// TIA Portal project "SortingStation" (V19)

(* hardware
DEVICE "S71500/ET200MP-Station_1"  S7-1500 station
   slot 0: "Profilschiene_0"  6ES7 590-1***0-0AA0
   slot 1: "PLC_1"  CPU 1511-1 PN  6ES7 511-1AK00-0AB0  V1.8
   slot 2: "AI 8xU/I/RTD/TC ST_1"  AI 8xU/I/RTD/TC ST  6ES7 531-7KF00-0AB0  V2.0
   slot 3: "AI 8xU/I/RTD/TC ST_2"  AI 8xU/I/RTD/TC ST  6ES7 531-7KF00-0AB0  V2.0
   slot 4: "AI 8xU/I/RTD/TC ST_3"  AI 8xU/I/RTD/TC ST  6ES7 531-7KF00-0AB0  V2.0
   slot 5: "AI 8xU/I/RTD/TC ST_4"  AI 8xU/I/RTD/TC ST  6ES7 531-7KF00-0AB0  V2.0
   slot 6: "DI 16x24VDC BA_1"  DI 16x24VDC BA  6ES7 521-1BH10-0AA0  V1.0
*)

// ===== PLC "PLC_1"  CPU 1511-1 PN =====

VAR_GLOBAL   // PLC tag table "Standard-Variablentabelle"
   "Tag_1" AT %I1.1 : Bool;
   "Tag_2" AT %Q1.6 : Bool;
   "Tag_3" AT %I1.2 : Bool;
END_VAR

VAR_GLOBAL   // PLC tag table "Tag table_1"
   "At exit" AT %I0.0 : Bool;
   "Start" AT %I0.1 : Bool;
   "Reset" AT %I0.2 : Bool;
   "Stop" AT %I0.3 : Bool;
   "Emergency stop" AT %I0.4 : Bool;
   "Auto" AT %I0.5 : Bool;
   "FACTORY I/O (Running)" AT %I0.6 : Bool;
   "Entry conveyor" AT %Q0.0 : Bool;
   "Stop blade" AT %Q0.1 : Bool;
   "Exit conveyor" AT %Q0.2 : Bool;
   "Sorter 1 turn" AT %Q0.3 : Bool;
   "Sorter 1 belt" AT %Q0.4 : Bool;
   "Sorter 2 turn" AT %Q0.5 : Bool;
   "Sorter 2 belt" AT %Q0.6 : Bool;
   "Sorter 3 turn" AT %Q0.7 : Bool;
   "Sorter 3 belt" AT %Q1.0 : Bool;
   "Start light" AT %Q1.1 : Bool;
   "Reset light" AT %Q1.2 : Bool;
   "Stop light" AT %Q1.3 : Bool;
   "Counter 1" AT %QD30 : DInt;
   "Counter 2" AT %QD34 : DInt;
   "Counter 3" AT %QD38 : DInt;
   "Vision sensor" AT %ID30 : DInt;
   "BoxLeft" AT %M0.1 : Bool;
   "BoxLeft2" AT %M0.2 : Bool;
   "BoxLeft3" AT %M0.4 : Bool;
   "SensorEdgeMem" AT %M0.0 : Bool;
   "BoxLeftStopBlade" AT %M0.3 : Bool;
   "Emitter" AT %Q1.4 : Bool;
END_VAR

DATA_BLOCK "EntryConveyor_DB"   // DB2
{ S7_Optimized_Access := 'TRUE' }
VERSION : 0.1
// stored: InstanceOfName Entry/ExitConveyor
"Entry/ExitConveyor"
BEGIN
END_DATA_BLOCK

DATA_BLOCK "Start/Stop_DB"   // DB3
{ S7_Optimized_Access := 'TRUE' }
VERSION : 0.1
// stored: InstanceOfName Start/Stop
"Start/Stop"
BEGIN
END_DATA_BLOCK

DATA_BLOCK "Stopblade_DB"   // DB4
{ S7_Optimized_Access := 'TRUE' }
VERSION : 0.1
// stored: InstanceOfName Stopblade
"Stopblade"
BEGIN
END_DATA_BLOCK

DATA_BLOCK "Sorter1_DB_1"   // DB5
{ S7_Optimized_Access := 'TRUE' }
VERSION : 0.1
// stored: InstanceOfName Sorter1
"Sorter1"
BEGIN
END_DATA_BLOCK

DATA_BLOCK "Sorter2_DB_1"   // DB8
{ S7_Optimized_Access := 'TRUE' }
VERSION : 0.1
// stored: InstanceOfName Sorter2
"Sorter2"
BEGIN
END_DATA_BLOCK

DATA_BLOCK "Sorter3_DB_1"   // DB9
{ S7_Optimized_Access := 'TRUE' }
VERSION : 0.1
// stored: InstanceOfName Sorter3
"Sorter3"
BEGIN
END_DATA_BLOCK

DATA_BLOCK "Counters_DB"   // DB11
{ S7_Optimized_Access := 'TRUE' }
VERSION : 0.1
// stored: InstanceOfName Counters
"Counters"
BEGIN
END_DATA_BLOCK

// folder: System blocks/Program resources

DATA_BLOCK "IEC_Timer_0_DB"   // DB1
{ S7_Optimized_Access := 'TRUE' }
AUTHOR : Simatic
FAMILY : IEC
NAME : IEC_TMR
VERSION : 1.0
// stored: InstanceOfName IEC_TIMER
"IEC_TIMER"
BEGIN
   PT := T#250MS;
END_DATA_BLOCK

DATA_BLOCK "IEC_Counter_1_DB"   // DB6
{ S7_Optimized_Access := 'TRUE' }
AUTHOR : Simatic
FAMILY : IEC
NAME : CNTR
VERSION : 1.0
// stored: InstanceOfName IEC_COUNTER
"IEC_COUNTER"
BEGIN
   PV := 100;
END_DATA_BLOCK

DATA_BLOCK "IEC_Counter_0_DB_1"   // DB7
{ S7_Optimized_Access := 'TRUE' }
AUTHOR : Simatic
FAMILY : IEC
NAME : CNTR
VERSION : 1.0
// stored: InstanceOfName IEC_COUNTER
"IEC_COUNTER"
BEGIN
   PV := 100;
END_DATA_BLOCK

DATA_BLOCK "IEC_Counter_2_DB"   // DB10
{ S7_Optimized_Access := 'TRUE' }
AUTHOR : Simatic
FAMILY : IEC
NAME : CNTR
VERSION : 1.0
// stored: InstanceOfName IEC_COUNTER
"IEC_COUNTER"
BEGIN
   PV := 100;
END_DATA_BLOCK

// folder: (top level)

FUNCTION_BLOCK "Start/Stop"   // FB1, LAD
{ S7_Optimized_Access := 'TRUE' }
VERSION : 0.1
BEGIN

REGION Network 1
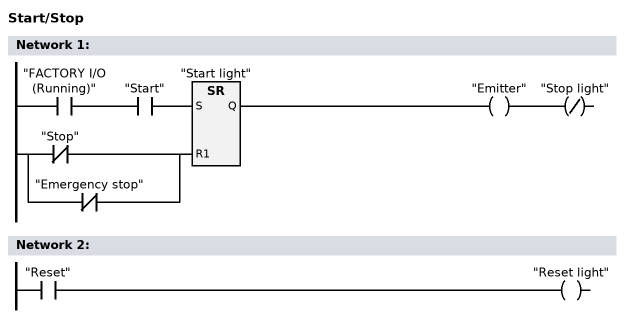
   RUNG wire#powerrail
      Contact( "FACTORY I/O (Running)" )
      Contact( "Start" )
      S_SR(operand := "Start light", r1 := wire#w1)
      Coil( "Emitter" )
      I_Coil( "Stop light" )
   END_RUNG
   RUNG wire#powerrail
      I_Contact( "Stop" )
   END_RUNG wire#w1
   RUNG wire#powerrail
      I_Contact( "Emergency stop" )
   END_RUNG wire#w1
   // the same network as SCL:
   IF "FACTORY I/O (Running)" AND "Start" THEN
       "Start light" := TRUE;   // SR flip-flop
   END_IF;
   IF NOT "Stop" OR NOT "Emergency stop" THEN "Start light" := FALSE; END_IF;
   "Emitter" := "Start light";
   "Stop light" := NOT "Start light";
END_REGION

REGION Network 2
   RUNG wire#powerrail
      Contact( "Reset" )
      Coil( "Reset light" )
   END_RUNG
   // the same network as SCL:
   "Reset light" := "Reset";
END_REGION
END_FUNCTION_BLOCK

FUNCTION_BLOCK "Sorter1"   // FB2, LAD
{ S7_Optimized_Access := 'TRUE' }
VERSION : 0.1
   VAR_TEMP   // added for the SCL form of the ladder/FBD networks
      _w1 : Bool;
   END_VAR
BEGIN

REGION Network 1
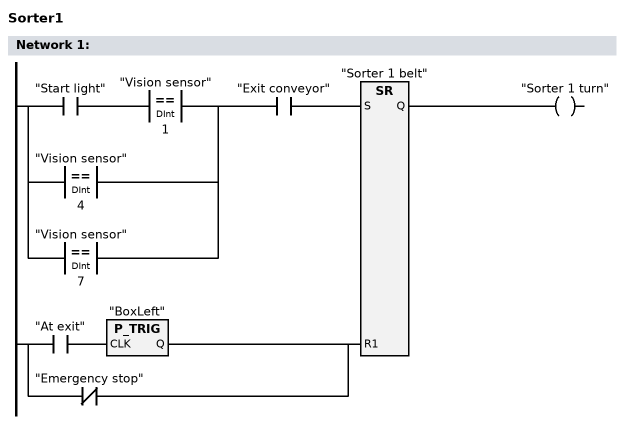
   RUNG wire#powerrail
      Contact( "Start light" )
      { S7_Templates := "SrcType := DInt" } EQ_Contact(in1 := "Vision sensor", in2 := 1)
      wire#w1
      Contact( "Exit conveyor" )
      S_SR(operand := "Sorter 1 belt", r1 := wire#w2)
      Coil( "Sorter 1 turn" )
   END_RUNG
   RUNG wire#powerrail
      { S7_Templates := "SrcType := DInt" } EQ_Contact(in1 := "Vision sensor", in2 := 4)
   END_RUNG wire#w1
   RUNG wire#powerrail
      { S7_Templates := "SrcType := DInt" } EQ_Contact(in1 := "Vision sensor", in2 := 7)
   END_RUNG wire#w1
   RUNG wire#powerrail
      Contact( "At exit" )
      P_Trig( "BoxLeft" )
   END_RUNG wire#w2
   RUNG wire#powerrail
      I_Contact( "Emergency stop" )
   END_RUNG wire#w2
   // the same network as SCL:
   #_w1 := "At exit" AND NOT "BoxLeft";   // rising edge
   "BoxLeft" := "At exit";
   IF (("Start light" AND ("Vision sensor" = 1)) OR ("Vision sensor" = 4) OR ("Vision sensor" = 7)) AND "Exit conveyor" THEN
       "Sorter 1 belt" := TRUE;   // SR flip-flop
   END_IF;
   IF #_w1 OR NOT "Emergency stop" THEN "Sorter 1 belt" := FALSE; END_IF;
   "Sorter 1 turn" := "Sorter 1 belt";
END_REGION
END_FUNCTION_BLOCK

FUNCTION_BLOCK "Sorter2"   // FB3, LAD
{ S7_Optimized_Access := 'TRUE' }
VERSION : 0.1
   VAR_TEMP   // added for the SCL form of the ladder/FBD networks
      _w1 : Bool;
   END_VAR
BEGIN

REGION Network 1
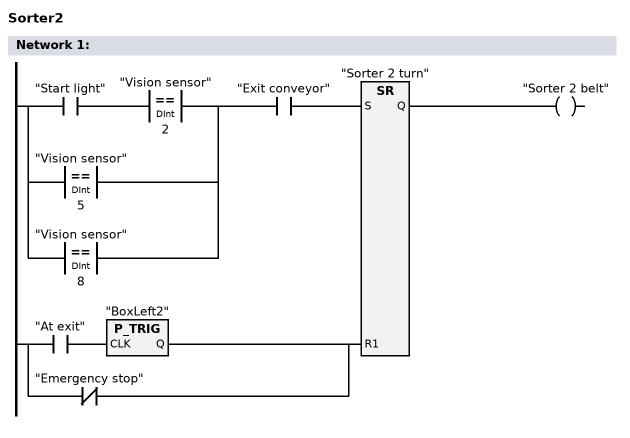
   RUNG wire#powerrail
      Contact( "Start light" )
      { S7_Templates := "SrcType := DInt" } EQ_Contact(in1 := "Vision sensor", in2 := 2)
      wire#w1
      Contact( "Exit conveyor" )
      S_SR(operand := "Sorter 2 turn", r1 := wire#w2)
      Coil( "Sorter 2 belt" )
   END_RUNG
   RUNG wire#powerrail
      { S7_Templates := "SrcType := DInt" } EQ_Contact(in1 := "Vision sensor", in2 := 5)
   END_RUNG wire#w1
   RUNG wire#powerrail
      { S7_Templates := "SrcType := DInt" } EQ_Contact(in1 := "Vision sensor", in2 := 8)
   END_RUNG wire#w1
   RUNG wire#powerrail
      Contact( "At exit" )
      P_Trig( "BoxLeft2" )
   END_RUNG wire#w2
   RUNG wire#powerrail
      I_Contact( "Emergency stop" )
   END_RUNG wire#w2
   // the same network as SCL:
   #_w1 := "At exit" AND NOT "BoxLeft2";   // rising edge
   "BoxLeft2" := "At exit";
   IF (("Start light" AND ("Vision sensor" = 2)) OR ("Vision sensor" = 5) OR ("Vision sensor" = 8)) AND "Exit conveyor" THEN
       "Sorter 2 turn" := TRUE;   // SR flip-flop
   END_IF;
   IF #_w1 OR NOT "Emergency stop" THEN "Sorter 2 turn" := FALSE; END_IF;
   "Sorter 2 belt" := "Sorter 2 turn";
END_REGION
END_FUNCTION_BLOCK

FUNCTION_BLOCK "Sorter3"   // FB4, LAD
{ S7_Optimized_Access := 'TRUE' }
VERSION : 0.1
   VAR_TEMP   // added for the SCL form of the ladder/FBD networks
      _w1 : Bool;
   END_VAR
BEGIN

REGION Network 1
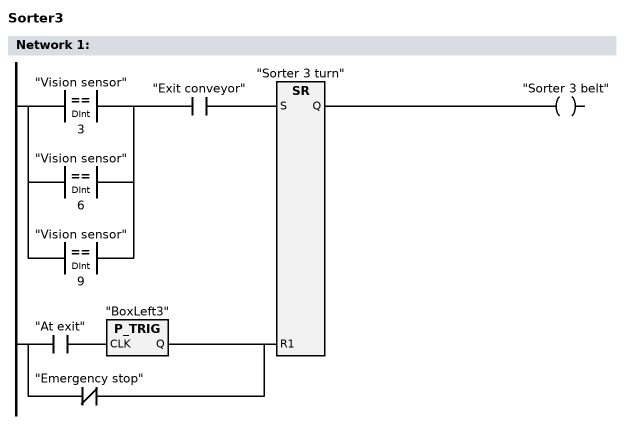
   RUNG wire#powerrail
      { S7_Templates := "SrcType := DInt" } EQ_Contact(in1 := "Vision sensor", in2 := 3)
      wire#w1
      Contact( "Exit conveyor" )
      S_SR(operand := "Sorter 3 turn", r1 := wire#w2)
      Coil( "Sorter 3 belt" )
   END_RUNG
   RUNG wire#powerrail
      { S7_Templates := "SrcType := DInt" } EQ_Contact(in1 := "Vision sensor", in2 := 6)
   END_RUNG wire#w1
   RUNG wire#powerrail
      { S7_Templates := "SrcType := DInt" } EQ_Contact(in1 := "Vision sensor", in2 := 9)
   END_RUNG wire#w1
   RUNG wire#powerrail
      Contact( "At exit" )
      P_Trig( "BoxLeft3" )
   END_RUNG wire#w2
   RUNG wire#powerrail
      I_Contact( "Emergency stop" )
   END_RUNG wire#w2
   // the same network as SCL:
   #_w1 := "At exit" AND NOT "BoxLeft3";   // rising edge
   "BoxLeft3" := "At exit";
   IF (("Vision sensor" = 3) OR ("Vision sensor" = 6) OR ("Vision sensor" = 9)) AND "Exit conveyor" THEN
       "Sorter 3 turn" := TRUE;   // SR flip-flop
   END_IF;
   IF #_w1 OR NOT "Emergency stop" THEN "Sorter 3 turn" := FALSE; END_IF;
   "Sorter 3 belt" := "Sorter 3 turn";
END_REGION
END_FUNCTION_BLOCK

FUNCTION_BLOCK "Stopblade"   // FB5, LAD
{ S7_Optimized_Access := 'TRUE' }
VERSION : 0.1
   VAR_TEMP   // added for the SCL form of the ladder/FBD networks
      _w1 : Bool;
      _w2 : Bool;
   END_VAR
BEGIN

REGION Network 1
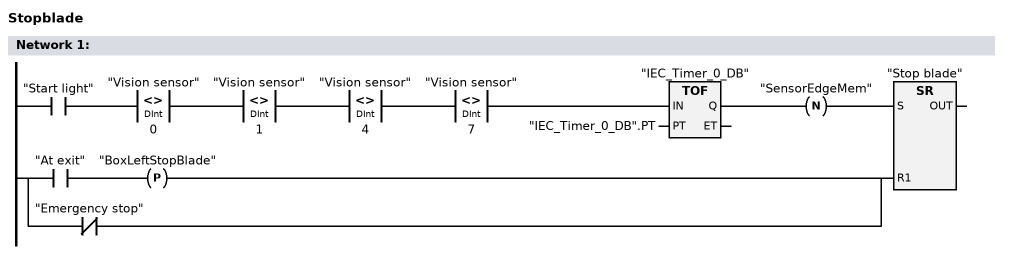
   "IEC_Timer_0_DB".TOF(IN := "Start light" AND ("Vision sensor" <> 0) AND ("Vision sensor" <> 1) AND ("Vision sensor" <> 4) AND ("Vision sensor" <> 7),
                        PT := "IEC_Timer_0_DB".PT);
   #_w1 := NOT "IEC_Timer_0_DB".Q AND "SensorEdgeMem";   // falling edge
   "SensorEdgeMem" := "IEC_Timer_0_DB".Q;
   #_w2 := "At exit" AND NOT "BoxLeftStopBlade";   // rising edge
   "BoxLeftStopBlade" := "At exit";
   IF #_w1 THEN
       "Stop blade" := TRUE;   // SR flip-flop
   END_IF;
   IF #_w2 OR NOT "Emergency stop" THEN "Stop blade" := FALSE; END_IF;
END_REGION
END_FUNCTION_BLOCK

FUNCTION_BLOCK "Entry/ExitConveyor"   // FB6, LAD
{ S7_Optimized_Access := 'TRUE' }
VERSION : 0.1
BEGIN

REGION Network 1
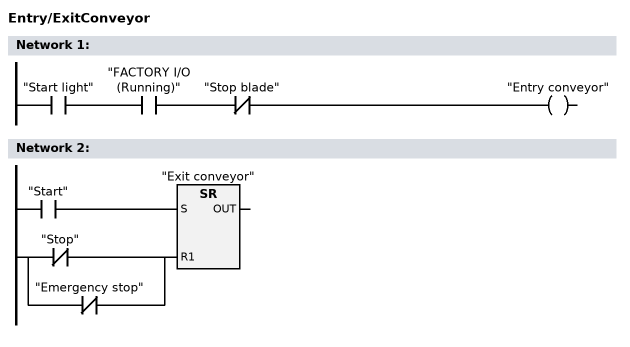
   RUNG wire#powerrail
      Contact( "Start light" )
      Contact( "FACTORY I/O (Running)" )
      I_Contact( "Stop blade" )
      Coil( "Entry conveyor" )
   END_RUNG
   // the same network as SCL:
   "Entry conveyor" := "Start light" AND "FACTORY I/O (Running)" AND NOT "Stop blade";
END_REGION

REGION Network 2
   RUNG wire#powerrail
      Contact( "Start" )
      S_SR(operand := "Exit conveyor", r1 := wire#w1)
   END_RUNG
   RUNG wire#powerrail
      I_Contact( "Stop" )
   END_RUNG wire#w1
   RUNG wire#powerrail
      I_Contact( "Emergency stop" )
   END_RUNG wire#w1
   // the same network as SCL:
   IF "Start" THEN
       "Exit conveyor" := TRUE;   // SR flip-flop
   END_IF;
   IF NOT "Stop" OR NOT "Emergency stop" THEN "Exit conveyor" := FALSE; END_IF;
END_REGION
END_FUNCTION_BLOCK

FUNCTION_BLOCK "Counters"   // FB7, LAD
{ S7_Optimized_Access := 'TRUE' }
VERSION : 0.1
BEGIN

REGION Network 1
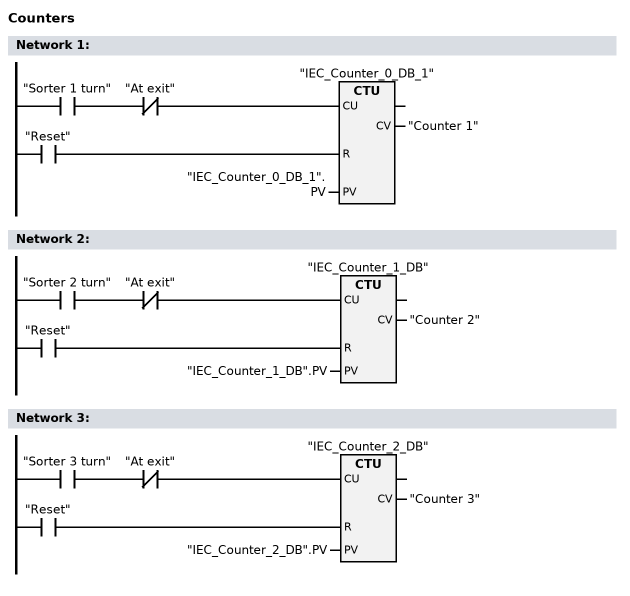
   "IEC_Counter_0_DB_1".CTU(CU := "Sorter 1 turn" AND NOT "At exit",
                           R := "Reset",
                           PV := "IEC_Counter_0_DB_1".PV,
                           CV => "Counter 1");
END_REGION

REGION Network 2
   "IEC_Counter_1_DB".CTU(CU := "Sorter 2 turn" AND NOT "At exit",
                          R := "Reset",
                          PV := "IEC_Counter_1_DB".PV,
                          CV => "Counter 2");
END_REGION

REGION Network 3
   "IEC_Counter_2_DB".CTU(CU := "Sorter 3 turn" AND NOT "At exit",
                          R := "Reset",
                          PV := "IEC_Counter_2_DB".PV,
                          CV => "Counter 3");
END_REGION
END_FUNCTION_BLOCK

FUNCTION "MHJ-PLC-Lab-Function-S71500" : Void   // FC9000, SCL
{ S7_Optimized_Access := 'TRUE' }
VERSION : 0.1
   VAR_TEMP
      Value : Byte;
      ForCounter : Int;
   END_VAR
   VAR CONSTANT
      Value_01_DW : DWord := 16#1223_5486;
      Value_02_DW : DWord := 16#A6C9_D1F5;
   END_VAR
BEGIN

   #Value:=PEEK(area := 16#82,
        dbNumber := 0,
        byteOffset := 511);
   #Value := #Value + 1;

   POKE(area := 16#82,
        dbNumber := 0,
        byteOffset := 511,
        value := #Value);

   POKE(area := 16#82,
        dbNumber := 0,
        byteOffset := 1016,
        value := #Value_01_DW);
   POKE(area := 16#82,
        dbNumber := 0,
        byteOffset := 1020,
        value := #Value_02_DW);

   FOR #ForCounter := 0 TO 63 DO
       #Value:=PEEK(area := 16#1,
            dbNumber := 0,
            byteOffset := #ForCounter);
       POKE(area := 16#81,
            dbNumber := 0,
            byteOffset := #ForCounter,
            value := #Value);
   END_FOR;
   #Value := PEEK(area := 16#1,
                  dbNumber := 0,
                  byteOffset := 512);
   POKE(area := 16#82,
        dbNumber := 0,
        byteOffset := 512,
        value := #Value);
END_FUNCTION

ORGANIZATION_BLOCK "Main"   // OB1, FBD, ProgramCycle
TITLE = "Main Program Sweep (Cycle)"
{ S7_Optimized_Access := 'TRUE' }
VERSION : 0.1
   VAR_INPUT
      Initial_Call : Bool;   // Initial call of this OB
      Remanence : Bool;   // =True, if remanent data are available
   END_VAR
   VAR_TEMP   // added for the SCL form of the ladder/FBD networks
      _w1 : Bool;
      _w2 : Bool;
      _w3 : Bool;
      _w4 : Bool;
      _w5 : Bool;
      _w6 : Bool;
   END_VAR
BEGIN

REGION Network 1
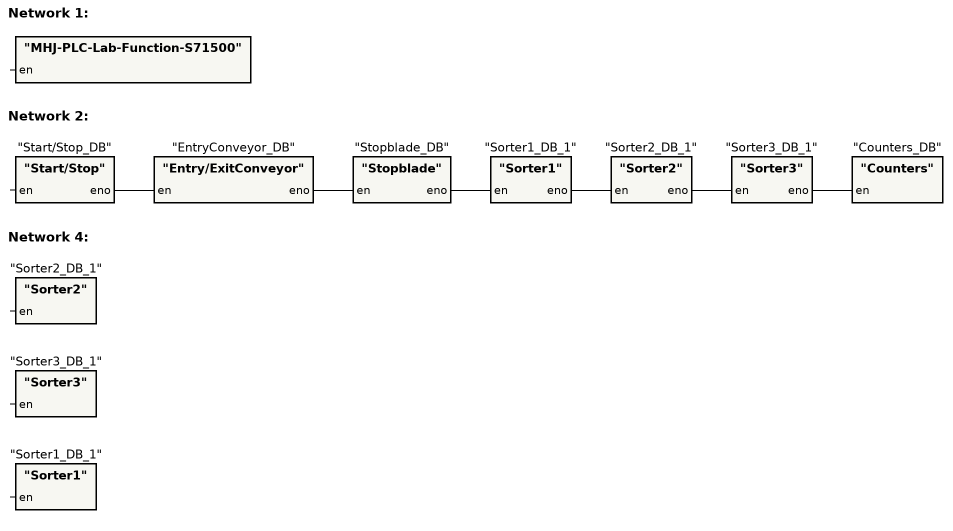
   "MHJ-PLC-Lab-Function-S71500"();
END_REGION

REGION Network 2
   "Start/Stop_DB"(ENO => #_w1);   // "Start/Stop"
   "EntryConveyor_DB"(EN := #_w1, ENO => #_w2);   // "Entry/ExitConveyor"
   "Stopblade_DB"(EN := #_w2, ENO => #_w3);   // "Stopblade"
   "Sorter1_DB_1"(EN := #_w3, ENO => #_w4);   // "Sorter1"
   "Sorter2_DB_1"(EN := #_w4, ENO => #_w5);   // "Sorter2"
   "Sorter3_DB_1"(EN := #_w5, ENO => #_w6);   // "Sorter3"
   IF #_w6 THEN
       "Counters_DB"();   // "Counters"
   END_IF;
END_REGION

REGION Network 4
   "Sorter2_DB_1"();   // "Sorter2"
   "Sorter3_DB_1"();   // "Sorter3"
   "Sorter1_DB_1"();   // "Sorter1"
END_REGION
END_ORGANIZATION_BLOCK